FUNCTION IsValidNode : BOOL
VAR_INPUT
	Node : I_Node;
END_VAR

IsValidNode := Node <> 0;

END_FUNCTION

(* stored: Version 1.1.0.1, ProductVersion 3.1.4024.12
   POU IsValidNode: Id {e61148da-078b-010d-0172-eeefce041b99}, SpecialFunc None *)
